// TIA Portal V19 export
TYPE "LAF_typeAxisDiagErrorWord"
TITLE = LAF_typeAxisDiagErrorWord
// Errors of a Technology Object
// stored: Access Published
   STRUCT
      bit00_SystemFault { ExternalWritable := 'False'} : Bool;   // A system-internal error has occurred / Enable
      bit01_ConfigFault { ExternalWritable := 'False'} : Bool;   // Configuration error. One or more configuration parameters are inconsistent or invalid / Error
      bit02_UserFault { ExternalWritable := 'False'} : Bool;   // Error in user program at a Motion Control instruction or its use / RestartActive
      bit03_CommandNotAccepted { ExternalWritable := 'False'} : Bool;   // Job cannot be executed. A Motion Control instruction cannot be executed because the necessary conditions have not been met / OnlineStartValuesChanged
      bit04_DriveFault { ExternalWritable := 'False'} : Bool;   // Error in drive / ControlPanelActive
      bit05_SensorFault { ExternalWritable := 'False'} : Bool;   // Error in encoder system / HomingDone
      bit06_DynamicError { ExternalWritable := 'False'} : Bool;   // Specified dynamic values are limited to permissible values / Done
      bit07_CommunicationFault { ExternalWritable := 'False'} : Bool;   // Missing or faulty communication / StandStill
      bit08_SWLimit { ExternalWritable := 'False'} : Bool;   // Software limit switch reached or overtraveled / PositioningCommand
      bit09_HWLimit { ExternalWritable := 'False'} : Bool;   // Hardware limit switch reached or overtraveled / JogCommand
      bit10_HomingError { ExternalWritable := 'False'} : Bool;   // Error during homing operation. The homing cannot be completed / VelocityCommand
      bit11_FollowingErrorFault { ExternalWritable := 'False'} : Bool;   // Following error limits exceeded / HomingCommand
      bit12_PositioningFault { ExternalWritable := 'False'} : Bool;   // Positioning error / ConstantVelocity
      bit13_PeripheralError { ExternalWritable := 'False'} : Bool;   // Error accessing a logical address / Accelerating
      bit14_SynchronousError { ExternalWritable := 'False'} : Bool;   // Error during synchronous operation. The leading axis specified in the Motion Control instruction was not configured as a possible leading axis / Decelerating
      bit15_AdaptionError { ExternalWritable := 'False'} : Bool;   // Error in automatic data transfer / SWLimitMinActive
      bit16_Reserved { ExternalWritable := 'False'} : Bool;   // Reserved / SWLimitMaxActive
      bit17_Reserved { ExternalWritable := 'False'} : Bool;   // Reserved / HWLimitMinActive
      bit18_Reserved { ExternalWritable := 'False'} : Bool;   // Reserved / HWLimitMaxActive
      bit19_Reserved { ExternalWritable := 'False'} : Bool;   // Reserved
      bit20_Reserved { ExternalWritable := 'False'} : Bool;   // Reserved
      bit21_Reserved { ExternalWritable := 'False'} : Bool;   // Reserved / Synchronizing
      bit22_Reserved { ExternalWritable := 'False'} : Bool;   // Reserved / Synhronous
      bit23_Reserved { ExternalWritable := 'False'} : Bool;   // Reserved / SuperimposedMotionCommand
      bit24_Reserved { ExternalWritable := 'False'} : Bool;   // Reserved / PhasingCommand
      bit25_Reserved { ExternalWritable := 'False'} : Bool;   // Reserved / AxisSimulation
      bit26_Reserved { ExternalWritable := 'False'} : Bool;   // Reserved / TorqueLimitingCommand
      bit27_Reserved { ExternalWritable := 'False'} : Bool;   // Reserved / InLimitation
      bit28_Reserved { ExternalWritable := 'False'} : Bool;   // Reserved / NonPositionControlled
      bit29_Reserved { ExternalWritable := 'False'} : Bool;   // Reserved
      bit30_Reserved { ExternalWritable := 'False'} : Bool;   // Reserved / InClamping
      bit31_Reserved { ExternalWritable := 'False'} : Bool;   // Reserved
   END_STRUCT;
END_TYPE
